KUKA KRL program: TEMPLATE.src, TEMPLATE.dat

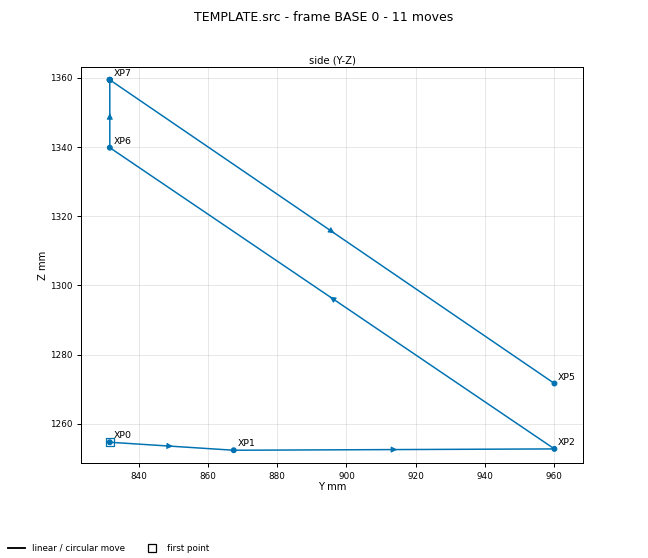
[picture p0: tool path of TEMPLATE.src in frame BASE 0, 11 of 12 moves have a stored position in this frame; points joined in program order, loops and branches not executed]
--- TEMPLATE.src ---
&ACCESS RVP
&REL 96
&PARAM TEMPLATE = C:\KRC\Roboter\Template\vorgabe
&PARAM EDITMASK = *
DEF TEMPLATE( )
;FOLD INI
  ;FOLD BASISTECH INI
    GLOBAL INTERRUPT DECL 3 WHEN $STOPMESS==TRUE DO IR_STOPM ( )
    INTERRUPT ON 3
    BAS (#INITMOV,0 )
  ;ENDFOLD (BASISTECH INI)
  ;FOLD USER INI
    ;Make your modifications here

  ;ENDFOLD (USER INI)
;ENDFOLD (INI)

;FOLD PTP HOME Vel=10 % DEFAULT;%{PE}%R 5.6.13,%MKUKATPBASIS,%CMOVE,%VPTP,%P 1:PTP, 2:HOME, 3:, 5:10, 7:DEFAULT
$BWDSTART=FALSE
PDAT_ACT=PDEFAULT
FDAT_ACT=FHOME
BAS(#PTP_PARAMS,10)
$H_POS=XHOME
PTP XHOME
;ENDFOLD
;FOLD LIN P0 Vel=0.1 m/s CPDAT4 Tool[1] Base[0];%{PE}%R 5.6.13,%MKUKATPBASIS,%CMOVE,%VLIN,%P 1:LIN, 2:P0, 3:, 5:0.1, 7:CPDAT4
$BWDSTART=FALSE
LDAT_ACT=LCPDAT4
FDAT_ACT=FP0
BAS(#CP_PARAMS,0.1)
LIN XP0
;ENDFOLD
;FOLD OUT 36 'Gas 2' State=TRUE CONT;%{PE}%R 5.6.13,%MKUKATPBASIS,%COUT,%VOUTX,%P 2:36, 3:Gas 2, 5:TRUE, 6:CONTINUE
CONTINUE
$OUT[36]=TRUE
;ENDFOLD
;FOLD ANOUT POWDER=0.2 ;%{PE}%R 5.6.13,%MKUKATPBASIS,%CANA,%VANOUT_STAT,%P 2:CHANNEL_1, 4:0.2
$ANOUT[1]=0.2
;ENDFOLD
;FOLD OUT 33 'Gas 1' State=TRUE CONT;%{PE}%R 5.6.13,%MKUKATPBASIS,%COUT,%VOUTX,%P 2:33, 3:Gas 1, 5:TRUE, 6:CONTINUE
CONTINUE
$OUT[33]=TRUE
;ENDFOLD
;FOLD WAIT Time=0.5 sec;%{PE}%R 5.6.13,%MKUKATPBASIS,%CWAIT,%VWAIT,%P 2:0.5
WAIT SEC 0.5
;ENDFOLD
;FOLD LIN P1 Vel=0.1 m/s CPDAT1 Tool[1] Base[0];%{PE}%R 5.6.13,%MKUKATPBASIS,%CMOVE,%VLIN,%P 1:LIN, 2:P1, 3:, 5:0.1, 7:CPDAT1
$BWDSTART=FALSE
LDAT_ACT=LCPDAT1
FDAT_ACT=FP1
BAS(#CP_PARAMS,0.1)
LIN XP1
;ENDFOLD
;FOLD SYN OUT 34 'Laser Shutter' State=TRUE at START Delay=0 ms;%{PE}%R 5.6.13,%MKUKATPBASIS,%COUT,%VSYNOUT,%P 2:34, 3:Laser Shutter, 5:TRUE, 7:0, 9:0, 12:0
TRIGGER WHEN DISTANCE=0 DELAY=0 DO $OUT[34]=TRUE
;ENDFOLD
;FOLD LIN P2 Vel=0.1 m/s CPDAT2 Tool[1] Base[0];%{PE}%R 5.6.13,%MKUKATPBASIS,%CMOVE,%VLIN,%P 1:LIN, 2:P2, 3:, 5:0.1, 7:CPDAT2
$BWDSTART=FALSE
LDAT_ACT=LCPDAT2
FDAT_ACT=FP2
BAS(#CP_PARAMS,0.1)
LIN XP2
;ENDFOLD
;FOLD LIN P6 Vel=0.1 m/s CPDAT6 Tool[1] Base[0];%{PE}%R 5.6.13,%MKUKATPBASIS,%CMOVE,%VLIN,%P 1:LIN, 2:P6, 3:, 5:0.1, 7:CPDAT6
$BWDSTART=FALSE
LDAT_ACT=LCPDAT6
FDAT_ACT=FP6
BAS(#CP_PARAMS,0.1)
LIN XP6
;ENDFOLD
;FOLD LIN P7 Vel=0.1 m/s CPDAT7 Tool[1] Base[0];%{PE}%R 5.6.13,%MKUKATPBASIS,%CMOVE,%VLIN,%P 1:LIN, 2:P7, 3:, 5:0.1, 7:CPDAT7
$BWDSTART=FALSE
LDAT_ACT=LCPDAT7
FDAT_ACT=FP7
BAS(#CP_PARAMS,0.1)
LIN XP7
;ENDFOLD
;FOLD LIN P8 Vel=0.1 m/s CPDAT8 Tool[1] Base[0];%{PE}%R 5.6.13,%MKUKATPBASIS,%CMOVE,%VLIN,%P 1:LIN, 2:P8, 3:, 5:0.1, 7:CPDAT8
$BWDSTART=FALSE
LDAT_ACT=LCPDAT8
FDAT_ACT=FP8
BAS(#CP_PARAMS,0.1)
LIN XP8
;ENDFOLD
;FOLD LIN P9 Vel=0.1 m/s CPDAT9 Tool[1] Base[0];%{PE}%R 5.6.13,%MKUKATPBASIS,%CMOVE,%VLIN,%P 1:LIN, 2:P9, 3:, 5:0.1, 7:CPDAT9
$BWDSTART=FALSE
LDAT_ACT=LCPDAT9
FDAT_ACT=FP9
BAS(#CP_PARAMS,0.1)
LIN XP9
;ENDFOLD
;FOLD LIN P10 Vel=0.1 m/s CPDAT10 Tool[1] Base[0];%{PE}%R 5.6.13,%MKUKATPBASIS,%CMOVE,%VLIN,%P 1:LIN, 2:P10, 3:, 5:0.1, 7:CPDAT10
$BWDSTART=FALSE
LDAT_ACT=LCPDAT10
FDAT_ACT=FP10
BAS(#CP_PARAMS,0.1)
LIN XP10
;ENDFOLD
;FOLD LIN P11 Vel=0.1 m/s CPDAT11 Tool[1] Base[0];%{PE}%R 5.6.13,%MKUKATPBASIS,%CMOVE,%VLIN,%P 1:LIN, 2:P11, 3:, 5:0.1, 7:CPDAT11
$BWDSTART=FALSE
LDAT_ACT=LCPDAT11
FDAT_ACT=FP11
BAS(#CP_PARAMS,0.1)
LIN XP11
;ENDFOLD
;FOLD LIN P12 Vel=0.1 m/s CPDAT12 Tool[1] Base[0];%{PE}%R 5.6.13,%MKUKATPBASIS,%CMOVE,%VLIN,%P 1:LIN, 2:P12, 3:, 5:0.1, 7:CPDAT12
$BWDSTART=FALSE
LDAT_ACT=LCPDAT12
FDAT_ACT=FP12
BAS(#CP_PARAMS,0.1)
LIN XP12
;ENDFOLD
;FOLD SYN OUT 34 'Laser Shutter' State=FALSE at START Delay=0 ms;%{PE}%R 5.6.13,%MKUKATPBASIS,%COUT,%VSYNOUT,%P 2:34, 3:Laser Shutter, 5:FALSE, 7:0, 9:0, 12:0
TRIGGER WHEN DISTANCE=0 DELAY=0 DO $OUT[34]=FALSE
;ENDFOLD
;FOLD SYN OUT 33 'Gas 1' State=FALSE at START Delay=0 ms;%{PE}%R 5.6.13,%MKUKATPBASIS,%COUT,%VSYNOUT,%P 2:33, 3:Gas 1, 5:FALSE, 7:0, 9:0, 12:0
TRIGGER WHEN DISTANCE=0 DELAY=0 DO $OUT[33]=FALSE
;ENDFOLD
;FOLD ANOUT POWDER=0 ;%{PE}%R 5.6.13,%MKUKATPBASIS,%CANA,%VANOUT_STAT,%P 2:CHANNEL_1, 4:0
$ANOUT[1]=0
;ENDFOLD
;FOLD SYN OUT 36 'Gas 2' State=FALSE at START Delay=0 ms;%{PE}%R 5.6.13,%MKUKATPBASIS,%COUT,%VSYNOUT,%P 2:36, 3:Gas 2, 5:FALSE, 7:0, 9:0, 12:0
TRIGGER WHEN DISTANCE=0 DELAY=0 DO $OUT[36]=FALSE
;ENDFOLD
;FOLD LIN P5 Vel=0.1 m/s CPDAT5 Tool[1] Base[0];%{PE}%R 5.6.13,%MKUKATPBASIS,%CMOVE,%VLIN,%P 1:LIN, 2:P5, 3:, 5:0.1, 7:CPDAT5
$BWDSTART=FALSE
LDAT_ACT=LCPDAT5
FDAT_ACT=FP5
BAS(#CP_PARAMS,0.1)
LIN XP5
;ENDFOLD
END

--- TEMPLATE.dat ---
&ACCESS RVP
&REL 96
&PARAM TEMPLATE = C:\KRC\Roboter\Template\vorgabe
&PARAM EDITMASK = *
DEFDAT  TEMPLATE
;FOLD EXTERNAL DECLARATIONS;%{PE}%MKUKATPBASIS,%CEXT,%VCOMMON,%P
;FOLD BASISTECH EXT;%{PE}%MKUKATPBASIS,%CEXT,%VEXT,%P
EXT  BAS (BAS_COMMAND  :IN,REAL  :IN )
DECL INT SUCCESS
;ENDFOLD (BASISTECH EXT)
;FOLD USER EXT;%{E}%MKUKATPUSER,%CEXT,%VEXT,%P
;Make here your modifications

;ENDFOLD (USER EXT)
;ENDFOLD (EXTERNAL DECLARATIONS)
DECL BASIS_SUGG_T LAST_BASIS={POINT1[] "P13                     ",POINT2[] "P14                     ",CP_PARAMS[] "CPDAT15                 ",PTP_PARAMS[] "PDAT0                   ",CONT[] "                        ",CP_VEL[] "0.1                     ",PTP_VEL[] "100                     ",SYNC_PARAMS[] "SYNCDAT                 ",SPL_NAME[] "S2                      "}
DECL E6POS XP1={X 984.648926,Y 867.426697,Z 1252.38098,A -157.865005,B 46.0220108,C -166.324295,S 2,T 35,E1 0.0,E2 0.0,E3 0.0,E4 0.0,E5 0.0,E6 0.0}
DECL FDAT FP1={TOOL_NO 1,BASE_NO 0,IPO_FRAME #BASE,POINT2[] " ",TQ_STATE FALSE}
DECL LDAT LCPDAT1={VEL 2.0,ACC 100.0,APO_DIST 100.0,APO_FAC 50.0,ORI_TYP #VAR,CIRC_TYP #BASE,JERK_FAC 50.0,EXAX_IGN 0}
DECL E6POS XP2={X 984.645325,Y 960.086487,Z 1252.76599,A -157.871094,B 46.0216713,C -166.328003,S 2,T 35,E1 0.0,E2 0.0,E3 0.0,E4 0.0,E5 0.0,E6 0.0}
DECL FDAT FP2={TOOL_NO 1,BASE_NO 0,IPO_FRAME #BASE,POINT2[] " ",TQ_STATE FALSE}
DECL LDAT LCPDAT2={VEL 2.0,ACC 100.0,APO_DIST 100.0,APO_FAC 50.0,ORI_TYP #VAR,CIRC_TYP #BASE,JERK_FAC 50.0,EXAX_IGN 0}
DECL E6POS XP3={X 984.630798,Y 831.62793,Z 1339.80701,A -157.880203,B 46.0213203,C -166.334702,S 2,T 35,E1 0.0,E2 0.0,E3 0.0,E4 0.0,E5 0.0,E6 0.0}
DECL FDAT FP3={TOOL_NO 1,BASE_NO 0,IPO_FRAME #BASE,POINT2[] " ",TQ_STATE FALSE}
DECL LDAT LCPDAT3={VEL 2.0,ACC 100.0,APO_DIST 100.0,APO_FAC 50.0,ORI_TYP #VAR,CIRC_TYP #BASE,JERK_FAC 50.0,EXAX_IGN 0}
DECL E6POS XP4={X 984.635925,Y 831.634888,Z 1359.40906,A -157.877594,B 46.0230103,C -166.333099,S 2,T 35,E1 0.0,E2 0.0,E3 0.0,E4 0.0,E5 0.0,E6 0.0}
DECL FDAT FP4={TOOL_NO 1,BASE_NO 0,IPO_FRAME #BASE,POINT2[] " ",TQ_STATE FALSE}
DECL LDAT LCPDAT4={VEL 2.0,ACC 100.0,APO_DIST 100.0,APO_FAC 50.0,ORI_TYP #VAR,CIRC_TYP #BASE,JERK_FAC 50.0,EXAX_IGN 0}
DECL E6POS XP0={X 984.636292,Y 831.612915,Z 1254.69397,A -157.876495,B 46.0204201,C -166.3311,S 2,T 35,E1 0.0,E2 0.0,E3 0.0,E4 0.0,E5 0.0,E6 0.0}
DECL FDAT FP0={TOOL_NO 1,BASE_NO 0,IPO_FRAME #BASE,POINT2[] " ",TQ_STATE FALSE}
DECL E6POS XP5={X 984.651123,Y 960.095581,Z 1271.66602,A -157.866699,B 46.0235291,C -166.325394,S 2,T 35,E1 0.0,E2 0.0,E3 0.0,E4 0.0,E5 0.0,E6 0.0}
DECL FDAT FP5={TOOL_NO 1,BASE_NO 0,IPO_FRAME #BASE,POINT2[] " ",TQ_STATE FALSE}
DECL LDAT LCPDAT5={VEL 2.0,ACC 100.0,APO_DIST 100.0,APO_FAC 50.0,ORI_TYP #VAR,CIRC_TYP #BASE,JERK_FAC 50.0,EXAX_IGN 0}
DECL LDAT LCPDAT6={VEL 2.0,ACC 100.0,APO_DIST 100.0,APO_FAC 50.0,ORI_TYP #VAR,CIRC_TYP #BASE,JERK_FAC 50.0,EXAX_IGN 0}
DECL E6POS XP6={X 984.630798,Y 831.62793,Z 1339.80701,A -157.880203,B 46.0213203,C -166.334702,S 2,T 35,E1 0.0,E2 0.0,E3 0.0,E4 0.0,E5 0.0,E6 0.0}
DECL FDAT FP6={TOOL_NO 1,BASE_NO 0,IPO_FRAME #BASE,POINT2[] " ",TQ_STATE FALSE}
DECL E6POS XP7={X 984.638184,Y 831.619324,Z 1359.40198,A -157.876099,B 46.0217209,C -166.331604,S 2,T 35,E1 0.0,E2 0.0,E3 0.0,E4 0.0,E5 0.0,E6 0.0}
DECL FDAT FP7={TOOL_NO 1,BASE_NO 0,IPO_FRAME #BASE,POINT2[] " ",TQ_STATE FALSE}
DECL LDAT LCPDAT7={VEL 2.0,ACC 100.0,APO_DIST 100.0,APO_FAC 50.0,ORI_TYP #VAR,CIRC_TYP #BASE,JERK_FAC 50.0,EXAX_IGN 0}
DECL E6POS XP8={X 984.638184,Y 831.619324,Z 1359.40198,A -157.876099,B 46.0217209,C -166.331604,S 2,T 35,E1 0.0,E2 0.0,E3 0.0,E4 0.0,E5 0.0,E6 0.0}
DECL FDAT FP8={TOOL_NO 1,BASE_NO 0,IPO_FRAME #BASE,POINT2[] " ",TQ_STATE FALSE}
DECL LDAT LCPDAT8={VEL 2.0,ACC 100.0,APO_DIST 100.0,APO_FAC 50.0,ORI_TYP #VAR,CIRC_TYP #BASE,JERK_FAC 50.0,EXAX_IGN 0}
DECL E6POS XP9={X 984.638184,Y 831.619324,Z 1359.40198,A -157.876099,B 46.0217209,C -166.331604,S 2,T 35,E1 0.0,E2 0.0,E3 0.0,E4 0.0,E5 0.0,E6 0.0}
DECL FDAT FP9={TOOL_NO 1,BASE_NO 0,IPO_FRAME #BASE,POINT2[] " ",TQ_STATE FALSE}
DECL LDAT LCPDAT9={VEL 2.0,ACC 100.0,APO_DIST 100.0,APO_FAC 50.0,ORI_TYP #VAR,CIRC_TYP #BASE,JERK_FAC 50.0,EXAX_IGN 0}
DECL E6POS XP10={X 984.638184,Y 831.619324,Z 1359.40198,A -157.876099,B 46.0217209,C -166.331604,S 2,T 35,E1 0.0,E2 0.0,E3 0.0,E4 0.0,E5 0.0,E6 0.0}
DECL FDAT FP10={TOOL_NO 1,BASE_NO 0,IPO_FRAME #BASE,POINT2[] " ",TQ_STATE FALSE}
DECL LDAT LCPDAT10={VEL 2.0,ACC 100.0,APO_DIST 100.0,APO_FAC 50.0,ORI_TYP #VAR,CIRC_TYP #BASE,JERK_FAC 50.0,EXAX_IGN 0}
DECL E6POS XP11={X 984.638184,Y 831.619324,Z 1359.40198,A -157.876099,B 46.0217209,C -166.331604,S 2,T 35,E1 0.0,E2 0.0,E3 0.0,E4 0.0,E5 0.0,E6 0.0}
DECL FDAT FP11={TOOL_NO 1,BASE_NO 0,IPO_FRAME #BASE,POINT2[] " ",TQ_STATE FALSE}
DECL LDAT LCPDAT11={VEL 2.0,ACC 100.0,APO_DIST 100.0,APO_FAC 50.0,ORI_TYP #VAR,CIRC_TYP #BASE,JERK_FAC 50.0,EXAX_IGN 0}
DECL E6POS XP12={X 984.638184,Y 831.619324,Z 1359.40198,A -157.876099,B 46.0217209,C -166.331604,S 2,T 35,E1 0.0,E2 0.0,E3 0.0,E4 0.0,E5 0.0,E6 0.0}
DECL FDAT FP12={TOOL_NO 1,BASE_NO 0,IPO_FRAME #BASE,POINT2[] " ",TQ_STATE FALSE}
DECL LDAT LCPDAT12={VEL 2.0,ACC 100.0,APO_DIST 100.0,APO_FAC 50.0,ORI_TYP #VAR,CIRC_TYP #BASE,JERK_FAC 50.0,EXAX_IGN 0}
DECL FDAT FS1={TOOL_NO 1,BASE_NO 0,IPO_FRAME #BASE,POINT2[] " ",TQ_STATE FALSE}
DECL LDAT LCPDAT13={VEL 2.0,ACC 100.0,APO_DIST 100.0,APO_FAC 50.0,ORI_TYP #VAR,CIRC_TYP #BASE,JERK_FAC 50.0,EXAX_IGN 0}
DECL E6POS XP13={X 984.642883,Y 831.616882,Z 1403.25305,A -157.879501,B 46.0230484,C -166.334198,S 2,T 35,E1 0.0,E2 0.0,E3 0.0,E4 0.0,E5 0.0,E6 0.0}
DECL E6POS XP14={X 984.643372,Y 859.865723,Z 1403.25098,A -157.879898,B 46.022831,C -166.334198,S 2,T 35,E1 0.0,E2 0.0,E3 0.0,E4 0.0,E5 0.0,E6 0.0}
DECL FDAT FP14={TOOL_NO 1,BASE_NO 0,IPO_FRAME #BASE,POINT2[] "XP13",TQ_STATE FALSE}
DECL LDAT LCPDAT14={VEL 2.0,ACC 100.0,APO_DIST 100.0,APO_FAC 50.0,ORI_TYP #VAR,CIRC_TYP #BASE,JERK_FAC 50.0,EXAX_IGN 0}
DECL LDAT CCPDAT14={CB {AUX_PT {ORI #CONSIDER,E1 #CONSIDER,E2 #CONSIDER,E3 #CONSIDER,E4 #CONSIDER,E5 #CONSIDER,E6 #CONSIDER},TARGET_PT {ORI #INTERPOLATE,E1 #INTERPOLATE,E2 #INTERPOLATE,E3 #INTERPOLATE,E4 #INTERPOLATE,E5 #INTERPOLATE,E6 #INTERPOLATE}}}
DECL FDAT FS2={TOOL_NO 1,BASE_NO 0,IPO_FRAME #BASE,POINT2[] " ",TQ_STATE FALSE}
DECL LDAT LCPDAT15={VEL 2.0,ACC 100.0,APO_DIST 100.0,APO_FAC 50.0,ORI_TYP #VAR,CIRC_TYP #BASE,JERK_FAC 50.0,EXAX_IGN 0}
DECL E6POS XP16={X 984.635193,Y 831.610291,Z 1394.78601,A -157.872299,B 46.0165596,C -166.327698,S 2,T 35,E1 0.0,E2 0.0,E3 0.0,E4 0.0,E5 0.0,E6 0.0}
ENDDAT
